TYPE T_Ctrl_SIf_AGS_Par :
STRUCT
END_STRUCT
END_TYPE

(* stored: Version 1.1.0.1, ProductVersion 3.1.0.26
   DUT T_Ctrl_SIf_AGS_Par: Id {db29b9c0-ab42-4364-8172-638ec7e45c0c} *)
